FUNCTION_BLOCK FB_CoE_BOOL EXTENDS FB_CoE_Base
VAR
	{attribute 'hide'}
	nValue : BOOL;
END_VAR

PROPERTY PROTECTED cbBufLen : UDINT
GET
cbBufLen := SIZEOF(nValue);
END_GET
END_PROPERTY

PROPERTY PROTECTED pSrcBuf : PVOID
GET
pSrcBuf := ADR(nValue);
END_GET
END_PROPERTY

{attribute 'monitoring':='call'}
PROPERTY Value : BOOL
GET
Value := nValue;
END_GET
SET
nValue := Value;

//Trigger a new write cycle
THIS^.bWriteDone 	:= FALSE;
END_SET
END_PROPERTY

END_FUNCTION_BLOCK

(* stored: Version 1.1.0.1, ProductVersion 3.1.4024.12
   POU FB_CoE_BOOL: Id {39f45e7f-99b3-4c6d-85c8-6844d97afae2}, SpecialFunc None
   Property cbBufLen: Id {0c3b03b7-8c5c-4263-ace7-67211946fa0d}
   Get Get: Id {58fd5a02-248a-45b5-b759-878688930a86}
   Property pSrcBuf: Id {ca7780d4-d12c-4c60-bb25-77e193818342}
   Get Get: Id {23feec92-1dc1-4516-8f37-7d87db9553af}
   Property Value: Id {9f999cbd-c82b-44b4-83d8-0ced22c86797}
   Get Get: Id {27a32eac-dcf3-4079-8c3e-be11721e5732}
   Set Set: Id {80186fa5-0caa-4310-9c1f-c5c11d17ab56} *)
